// TwinCAT 3 PLC project PLC2
// ProgramVersion: 3.1.4020.2
// libraries:
//   Tc2_Standard, * (Beckhoff Automation GmbH)
//   Tc2_System, * (Beckhoff Automation GmbH)
//   Tc3_Module, * (Beckhoff Automation GmbH)
// project tree:
//   DUTs/ ST_APIBetweenPLC.TcDUT
//   / PlcTask.TcTTO
//   POUs/ MAIN_852.TcPOU
// (motion and I/O tree: see PLC project plc1)
// real-time tasks:
//   TASK PlcTask: cycle T#10ms, priority 20, ADS port 350

CONFIGURATION PLC2
    RESOURCE PLC ON TwinCAT3
        TASK PlcTask(INTERVAL := T#10ms, PRIORITY := 20);
        PROGRAM MAIN_852 WITH PlcTask : MAIN_852;
    END_RESOURCE
END_CONFIGURATION

// ---- DUTs/ST_APIBetweenPLC.TcDUT
TYPE ST_APIBetweenPLC :
STRUCT
	_word: WORD;
	_int:INT;
	_Byte:BYTE;
	_String:STRING;
	_Bool:BOOL;
END_STRUCT
END_TYPE

// ---- POUs/MAIN_852.TcPOU
PROGRAM MAIN_852
VAR
	_ST_APIBetweenPLCRx AT%MW0: ST_APIBetweenPLC;
	_ST_APIBetweenPLCTx : ST_APIBetweenPLC;
	fbADSWRITE: ADSWRITE;
	Trig: Ton;
	sNetIdOfThOtherTCsystem: STRING :='10.122.128.1.1.1';
END_VAR

Trig(in:=NOT trig.Q ,PT:=T#500MS);
IF Trig.Q THEN
	_ST_APIBetweenPLCTx._int:=_ST_APIBetweenPLCTx._int+1;
END_IF
_ST_APIBetweenPLCTx._String:=concat('Value=', INT_TO_STRING(_ST_APIBetweenPLCTx._int));
fbADSWRITE(
	NETID:=sNetIdOfThOtherTCsystem , 
	PORT:=851 , 
	IDXGRP:=16#4020 , 
	IDXOFFS:=16#0 ,
 	LEN:=SIZEOF(_ST_APIBetweenPLCTx) , 
	SRCADDR:=ADR(_ST_APIBetweenPLCTx) ,
	WRITE:=Trig.Q , 
	TMOUT:= , 
	BUSY=> , 
	ERR=> , 
	ERRID=> );

END_PROGRAM
